(* CODESYS project Mahle_FilterLine_TempControl_17_01_20.project
   Title: Mahle_FilterLine_TempControl_03_01_20
   Version: 0.0.0.0

Project tree, tasks and I/O mapping:
  MyController : TM218LDAE24DRHN, Schneider Electric, order no. TM218LDAE24DRHN, version 4.0.1.26
      settings: Expansion Tasks.Expansion 1 Task Name = 'MAST'
    application Application
      libraries: Standard, * (System)
      task MAST (cyclic, interval 20 ms, priority 15, watchdog 100 ms x 1) calls POU
      function HiddenPOU [ST]
      global variables GVL
      program POU [FBD]
      function block tempAvergaging [ST]
      function block tempController [ST]
      function block calculateCycleTime [ST]
      function CheckBounds [ST]
      function block pressureAlarm [ST]
    Embedded Functions
      IO : IO, Schneider Electric, version 4.0.1.26
          input  iwIO_IW0 : WORD  // IW0
          input  iAuto : BOOL  // IW0.I0
          input  iPanelPB : BOOL  // IW0.I1
          input  iStartPB : BOOL  // IW0.I2
          input  iStopPB : BOOL  // IW0.I3
          input  iThyristorTrip : BOOL  // IW0.I6
          input  iFwdSensor : BOOL  // IW0.I8
          output qStartMC : BOOL  // QW0.Q0
          output qHeaterDown : BOOL  // QW0.Q1
          output qYellow : BOOL  // QW0.Q2
          output qGreen : BOOL  // QW0.Q3
          output qRed : BOOL  // QW0.Q4
          output qHooter : BOOL  // QW0.Q5
          unmapped channels: QW0
      HSC : HSC, Schneider Electric, version 4.0.1.26
    Serial Line 1
      SoMachine_Network_Manager : SoMachine-Network Manager, Schneider Electric, version 4.0.0.2
    Serial Line 2
      Modbus_Manager : Modbus Manager, Schneider Electric, version 4.0.0.2
    Ethernet
        settings: IPAddress = [192, 168, 1, 1]; SubnetMask = [255, 255, 255, 0]; WebServer = FALSE; FTP Server = FALSE; SoMachine Protocol = TRUE; Modbus Server = TRUE; NetManage Protocol = FALSE; SNMP protocol = FALSE; Enable Routing = FALSE
    Module_1 : TM2AMM3HT, Schneider Electric, order no. TM2AMM3HT, version 4.0.1.26
        settings: IW0.Maximum = 4000; IW1.Maximum = 1000; QW0.Maximum = 1000
        input  iwTempSensor : INT  // IW0
        input  iwPressureSensor : INT  // IW1
        output qwHeater : INT  // QW0
*)

// MyController/Application/GVL
VAR_GLOBAL
	thyristorTrip AT %MX600.0: BOOL;
	autoSel AT %MX600.1: BOOL;
	mcRunning AT %MX600.2: BOOL;
	heaterDown AT %MX600.3: BOOL;
	startSensing AT %MX600.4: BOOL;
	pressureLow AT %MX600.5: BOOL;
	resetPressMinMax AT %MX600.6: BOOL;
	cycleError AT %MX600.7: BOOL;
	startMCRun: BOOL;
	
	pressLowAlarm: BOOL;
	pressHighAlarm: BOOL;
END_VAR
VAR_GLOBAL RETAIN
	tempOffset AT %MD0: REAL :=0;
	puckTemp AT %MD1: REAL;
	finalCount AT %MD2: DINT;
	propGain AT %MD3: REAL;
	integGain AT %MD4: REAL;
	derivative AT %MD5: REAL;
	setTemp AT %MD6: REAL :=195;
	puckTempAvg AT %MD7: REAL;
	heaterManualSP AT %MD8: REAL :=50;
	heaterPIDOut AT %MD9: REAL;
	
	cycleTime AT %MD10: REAL;
	timeBWPucks AT %MD11: REAL;
	heaterLowRun AT %MD12: REAL :=48;
	heaterHighRun AT %MD13: REAL :=55;
	
	pressure AT %MD14: REAL;
	pressHighSet AT %MD15: REAL;
	pressLowSet AT %MD16: REAL;
	pressMin AT %MD17: REAL;
	pressMax AT %MD18: REAL;	
	pressureOffset AT %MD19: REAL;
	AvgPressure AT %MD21: REAL;
	
	startDelay AT %MW100: INT :=6;
	mcStopTime AT %MW101: INT :=30;
	pressAlarmDelay AT %MW102: INT;
	
	heaterManualOn AT %MX602.0: BOOL;
	heaterManualDown AT %MX602.1: BOOL;
	
END_VAR

// MyController/Application/POU
PROGRAM POU
VAR
	puckTemp1: REAL;
	tempAvergaging_0: tempAvergaging;
	PID_0: PID;
	RS_0: RS;
	runMC: BOOL;
	R_TRIG_0: R_TRIG;
	PID_1: PID_FIXCYCLE;
	TON_0: TON;
	tempController_0: tempController;
	TP_0: TP;
	mcStartDelayTime: TIME;
	TON_1: TON;
	calculateCycleTime_0: calculateCycleTime;
	sensorTrig: BOOL;
	TP_1: TP;
	stopTime: TIME;
	TON_2: TON;
	stopTimeET: TIME;
	stopHeater: BOOL;
	pressureAlarm_0: pressureAlarm;
	pressAlarm: BOOL;
	startProduction: BOOL;
	greenCont: BOOL;
	BLINK_0: BLINK;
	BLINK_1: BLINK;
	stopHeater1: BOOL;
	RS_1: RS;
END_VAR

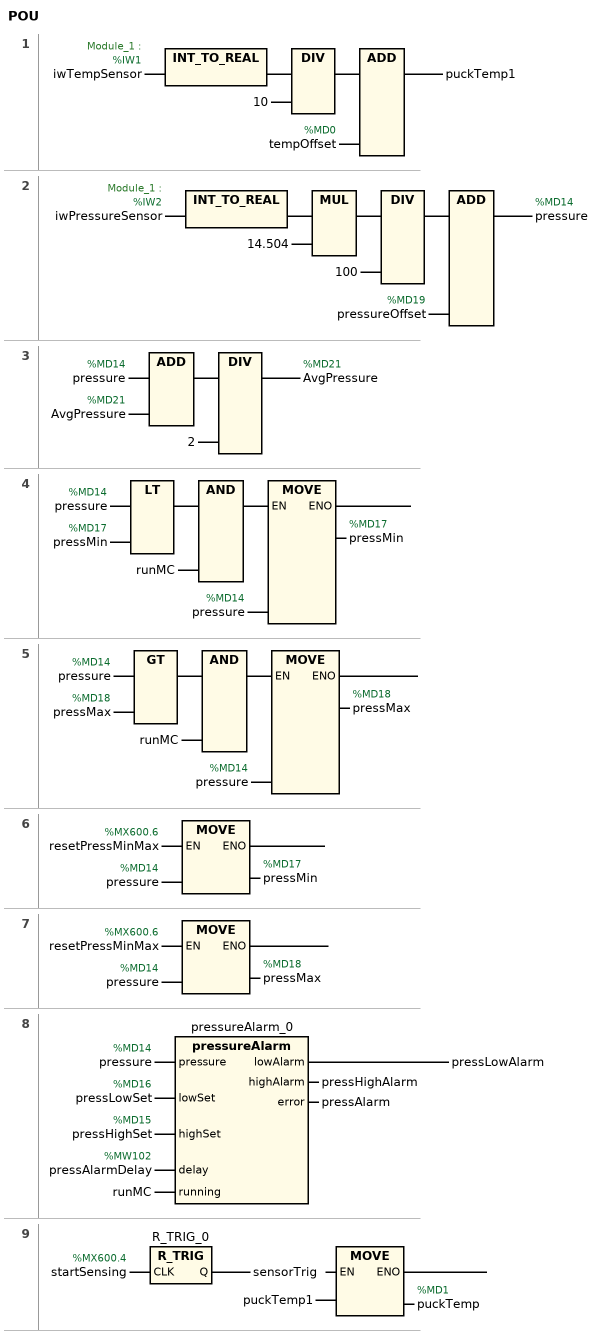
// NETWORK 1
//   iwTempSensor: Module_1 : | AT %IW1
//   tempOffset: AT %MD0
puckTemp1 := INT_TO_REAL(iwTempSensor) / 10 + tempOffset;

// NETWORK 2
//   iwPressureSensor: Module_1 : | AT %IW2
//   pressureOffset: AT %MD19
//   pressure: AT %MD14
pressure := (INT_TO_REAL(iwPressureSensor) * 14.504) / 100 + pressureOffset;

// NETWORK 3
//   pressure: AT %MD14
//   AvgPressure: AT %MD21
AvgPressure := (pressure + AvgPressure) / 2;

// NETWORK 4
//   pressure: AT %MD14
//   pressMin: AT %MD17
IF pressure < pressMin AND runMC THEN pressMin := pressure; END_IF

// NETWORK 5
//   pressure: AT %MD14
//   pressMax: AT %MD18
IF pressure > pressMax AND runMC THEN pressMax := pressure; END_IF

// NETWORK 6
//   resetPressMinMax: AT %MX600.6
//   pressure: AT %MD14
//   pressMin: AT %MD17
IF resetPressMinMax THEN pressMin := pressure; END_IF

// NETWORK 7
//   resetPressMinMax: AT %MX600.6
//   pressure: AT %MD14
//   pressMax: AT %MD18
IF resetPressMinMax THEN pressMax := pressure; END_IF

// NETWORK 8
//   pressure: AT %MD14
//   pressLowSet: AT %MD16
//   pressHighSet: AT %MD15
//   pressAlarmDelay: AT %MW102
pressureAlarm_0(
    pressure := pressure,
    lowSet := pressLowSet,
    highSet := pressHighSet,
    delay := pressAlarmDelay,
    running := runMC,
    highAlarm => pressHighAlarm,
    error => pressAlarm); // pressureAlarm
pressLowAlarm := pressureAlarm_0.lowAlarm;

// NETWORK 9
//   startSensing: AT %MX600.4
//   puckTemp: AT %MD1
R_TRIG_0(CLK := startSensing); // R_TRIG
sensorTrig := R_TRIG_0.Q;
IF R_TRIG_0.Q THEN puckTemp := puckTemp1; END_IF

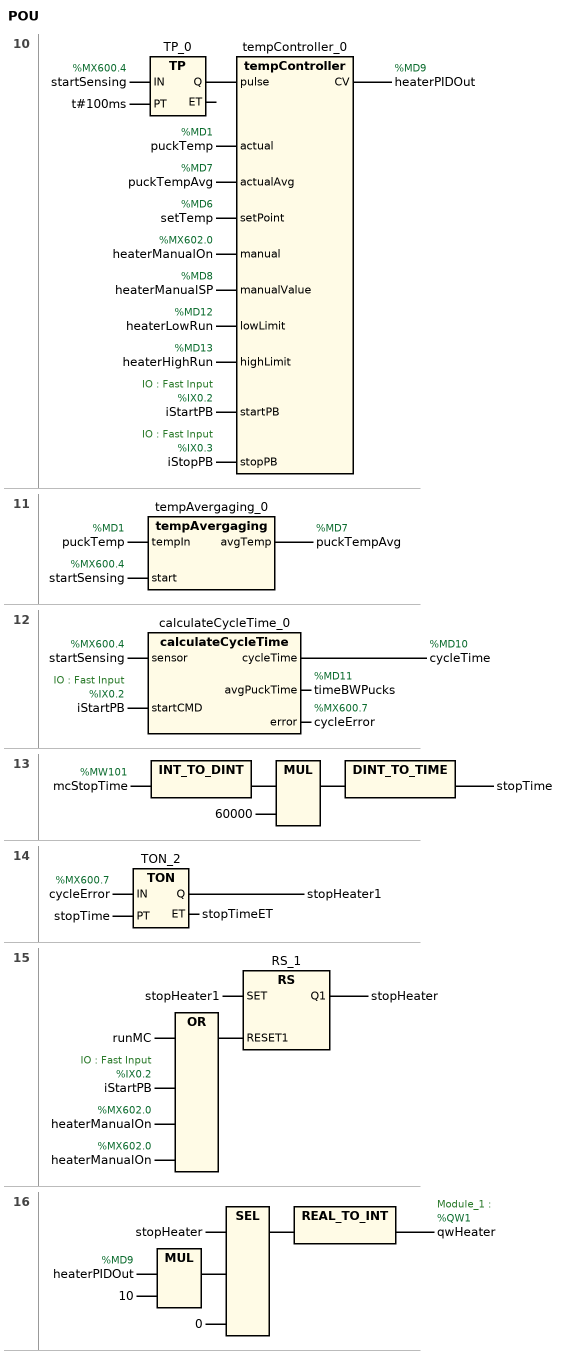
// NETWORK 10
//   startSensing: AT %MX600.4
//   puckTemp: AT %MD1
//   puckTempAvg: AT %MD7
//   setTemp: AT %MD6
//   heaterManualOn: AT %MX602.0
//   heaterManualSP: AT %MD8
//   heaterLowRun: AT %MD12
//   heaterHighRun: AT %MD13
//   iStartPB: IO : Fast Input | AT %IX0.2
//   iStopPB: IO : Fast Input | AT %IX0.3
//   heaterPIDOut: AT %MD9
TP_0(IN := startSensing, PT := t#100ms); // TP
tempController_0(
    pulse := TP_0.Q,
    actual := puckTemp,
    actualAvg := puckTempAvg,
    setPoint := setTemp,
    manual := heaterManualOn,
    manualValue := heaterManualSP,
    lowLimit := heaterLowRun,
    highLimit := heaterHighRun,
    startPB := iStartPB,
    stopPB := iStopPB); // tempController
heaterPIDOut := tempController_0.CV;

// NETWORK 11
//   puckTemp: AT %MD1
//   startSensing: AT %MX600.4
//   puckTempAvg: AT %MD7
tempAvergaging_0(tempIn := puckTemp, start := startSensing); // tempAvergaging
puckTempAvg := tempAvergaging_0.avgTemp;

// NETWORK 12
//   startSensing: AT %MX600.4
//   iStartPB: IO : Fast Input | AT %IX0.2
//   timeBWPucks: AT %MD11
//   cycleError: AT %MX600.7
//   cycleTime: AT %MD10
calculateCycleTime_0(
    sensor := startSensing,
    startCMD := iStartPB,
    avgPuckTime => timeBWPucks,
    error => cycleError); // calculateCycleTime
cycleTime := calculateCycleTime_0.cycleTime;

// NETWORK 13
//   mcStopTime: AT %MW101
stopTime := DINT_TO_TIME(INT_TO_DINT(mcStopTime) * 60000);

// NETWORK 14
//   cycleError: AT %MX600.7
TON_2(IN := cycleError, PT := stopTime, ET => stopTimeET); // TON
stopHeater1 := TON_2.Q;

// NETWORK 15
//   iStartPB: IO : Fast Input | AT %IX0.2
//   heaterManualOn: AT %MX602.0
RS_1(SET := stopHeater1, RESET1 := runMC OR iStartPB OR heaterManualOn OR heaterManualOn); // RS
stopHeater := RS_1.Q1;

// NETWORK 16
//   heaterPIDOut: AT %MD9
//   qwHeater: Module_1 : | AT %QW1
qwHeater := REAL_TO_INT(SEL(stopHeater, heaterPIDOut * 10, 0));

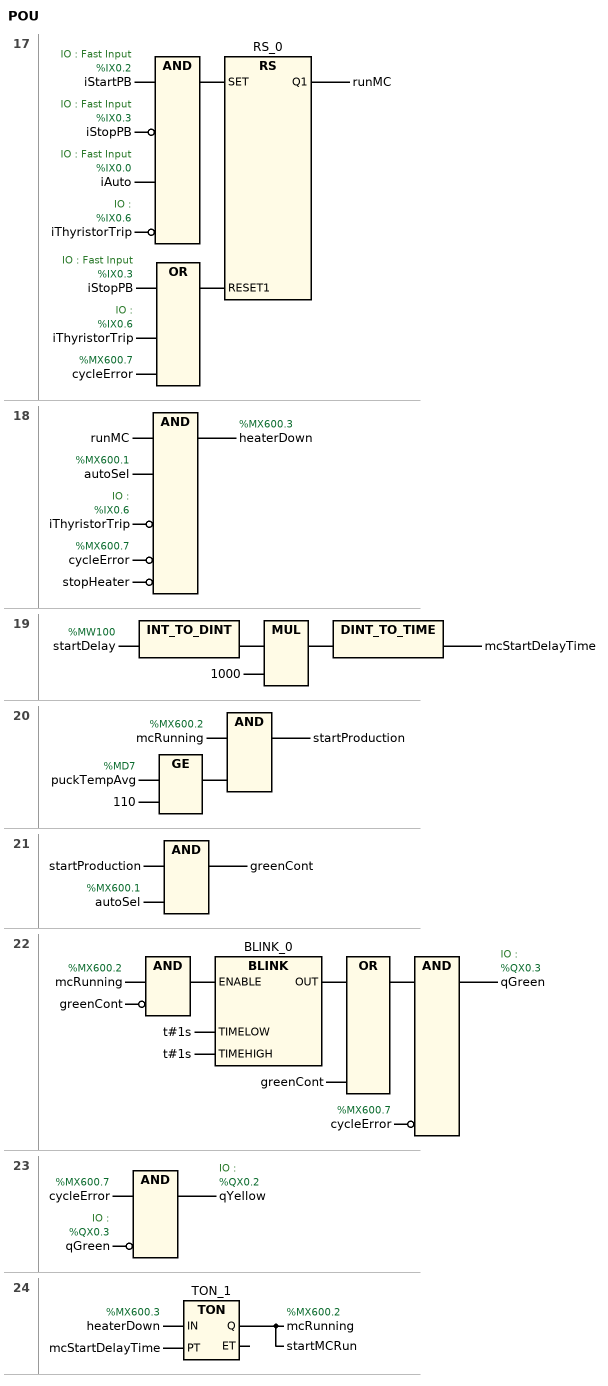
// NETWORK 17
//   iStartPB: IO : Fast Input | AT %IX0.2
//   iStopPB: IO : Fast Input | AT %IX0.3
//   iAuto: IO : Fast Input | AT %IX0.0
//   iThyristorTrip: IO : | AT %IX0.6
//   cycleError: AT %MX600.7
RS_0(SET := iStartPB AND NOT iStopPB AND iAuto AND NOT iThyristorTrip, RESET1 := iStopPB OR iThyristorTrip OR cycleError); // RS
runMC := RS_0.Q1;

// NETWORK 18
//   autoSel: AT %MX600.1
//   iThyristorTrip: IO : | AT %IX0.6
//   cycleError: AT %MX600.7
//   heaterDown: AT %MX600.3
heaterDown := runMC AND autoSel AND NOT iThyristorTrip AND NOT cycleError AND NOT stopHeater;

// NETWORK 19
//   startDelay: AT %MW100
mcStartDelayTime := DINT_TO_TIME(INT_TO_DINT(startDelay) * 1000);

// NETWORK 20
//   mcRunning: AT %MX600.2
//   puckTempAvg: AT %MD7
startProduction := mcRunning AND puckTempAvg >= 110;

// NETWORK 21
//   autoSel: AT %MX600.1
greenCont := startProduction AND autoSel;

// NETWORK 22
//   mcRunning: AT %MX600.2
//   cycleError: AT %MX600.7
//   qGreen: IO : | AT %QX0.3
BLINK_0(ENABLE := mcRunning AND NOT greenCont, TIMELOW := t#1s, TIMEHIGH := t#1s); // BLINK
qGreen := (BLINK_0.OUT OR greenCont) AND NOT cycleError;

// NETWORK 23
//   cycleError: AT %MX600.7
//   qGreen: IO : | AT %QX0.3
//   qYellow: IO : | AT %QX0.2
qYellow := cycleError AND NOT qGreen;

// NETWORK 24
//   heaterDown: AT %MX600.3
//   mcRunning: AT %MX600.2
TON_1(IN := heaterDown, PT := mcStartDelayTime); // TON
mcRunning := TON_1.Q;
startMCRun := TON_1.Q;

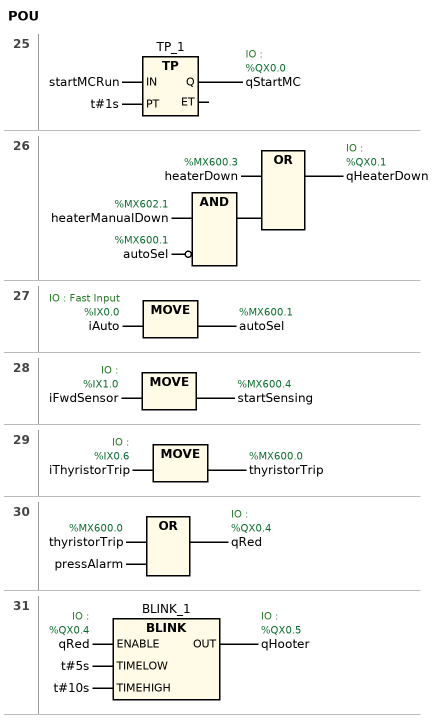
// NETWORK 25
//   qStartMC: IO : | AT %QX0.0
TP_1(IN := startMCRun, PT := t#1s); // TP
qStartMC := TP_1.Q;

// NETWORK 26
//   heaterDown: AT %MX600.3
//   heaterManualDown: AT %MX602.1
//   autoSel: AT %MX600.1
//   qHeaterDown: IO : | AT %QX0.1
qHeaterDown := heaterDown OR heaterManualDown AND NOT autoSel;

// NETWORK 27
//   iAuto: IO : Fast Input | AT %IX0.0
//   autoSel: AT %MX600.1
autoSel := iAuto;

// NETWORK 28
//   iFwdSensor: IO : | AT %IX1.0
//   startSensing: AT %MX600.4
startSensing := iFwdSensor;

// NETWORK 29
//   iThyristorTrip: IO : | AT %IX0.6
//   thyristorTrip: AT %MX600.0
thyristorTrip := iThyristorTrip;

// NETWORK 30
//   thyristorTrip: AT %MX600.0
//   qRed: IO : | AT %QX0.4
qRed := thyristorTrip OR pressAlarm;

// NETWORK 31
//   qRed: IO : | AT %QX0.4
//   qHooter: IO : | AT %QX0.5
BLINK_1(ENABLE := qRed, TIMELOW := t#5s, TIMEHIGH := t#10s); // BLINK
qHooter := BLINK_1.OUT;

END_PROGRAM

// MyController/Application/pressureAlarm
FUNCTION_BLOCK pressureAlarm
VAR_INPUT
	pressure: REAL;
	lowSet: REAL;
	highSet: REAL;
	delay: INT;
	running: BOOL;
END_VAR
VAR_OUTPUT
	lowAlarm: BOOL;
	highAlarm: BOOL;
	error: BOOL;
END_VAR
VAR
	timeDelay: TIME;
	startTON1: BOOL;
	startTON2: BOOL;
	TON1: TON;
	TON2: TON;
END_VAR

timeDelay := DINT_TO_TIME(INT_TO_DINT(delay)*1000);

TON1(IN:=startTON1, PT:=timeDelay);
TON2(IN:=startTON2, PT:=timeDelay);

IF running THEN
	IF pressure < lowSet THEN
		startTON1 := TRUE;
	ELSE
		startTON1 := FALSE;
	END_IF

	IF pressure > highSet THEN
		startTON2 := TRUE;
	ELSE
		startTON2 := FALSE;
	END_IF			
	
	IF ton1.Q THEN
		lowAlarm := TRUE;
	ELSE
		lowAlarm := FALSE;
	END_IF
	
	IF ton2.Q THEN
		highAlarm := TRUE;
	ELSE
		highAlarm := FALSE;
	END_IF
	
	IF lowAlarm OR highAlarm THEN
		error := TRUE;
	ELSE
		error := FALSE;
	END_IF
END_IF

END_FUNCTION_BLOCK

// MyController/Application/tempController
FUNCTION_BLOCK tempController
VAR_INPUT
	pulse: BOOL;
	actual: REAL;
	actualAvg: REAL;
	setPoint: REAL;
	manual: BOOL;
	manualValue: REAL;
	lowLimit: REAL;
	highLimit: REAL;
	startPB: BOOL;
	stopPB: BOOL;
END_VAR
VAR_OUTPUT
	CV: REAL;
END_VAR
VAR
	error: REAL;
	errorPC: REAL;
	CV1: REAL;
	errorPCAbs: REAL;
	errorFromAvg: REAL;
	startHeater: BOOL;
	CV2: REAL;
END_VAR

IF startPB AND NOT manual THEN
	startHeater := TRUE;
	CV1 := highLimit;
END_IF
IF pulse AND NOT manual THEN
	error := setPoint - actual;
	errorPC := (error*100)/setPoint;
	errorFromAvg := actualAvg - actual;
	IF errorFromAvg < 20 AND errorFromAvg > -20 THEN
	
		IF errorPC >=0 THEN
			errorPCAbs := errorPC;
		ELSE
			errorPCAbs := -1*errorPC;
		END_IF
	
		IF errorPCAbs < 2 THEN
			CV1 := CV+(errorPC/90);
		ELSIF errorPCAbs < 5 THEN
			CV1 := CV + (errorPC/50);
		ELSIF errorPCAbs < 15 THEN
			CV1 := CV + (errorPC/75);
		ELSE
			CV1 := CV + (errorPC/100);				
		END_IF
	END_IF
END_IF

IF manual THEN
	CV := manualValue;
ELSE
	CV := CV2;
END_IF

IF CV1 < lowLimit THEN
	CV2 := lowLimit;
ELSIF CV1 > highLimit THEN
	CV2 := highLimit;
ELSE
	CV2 := CV1;
END_IF

END_FUNCTION_BLOCK

// MyController/Application/tempAvergaging
FUNCTION_BLOCK tempAvergaging
VAR_INPUT
	tempIn: REAL;
	start: BOOL;
END_VAR
VAR_OUTPUT
	avgTemp: REAL;
END_VAR
VAR
	counter1: CTU;
	x1: REAL :=0;
	x2: REAL :=0;
	x3: REAL :=0;
	x4: REAL :=0;
	x5: REAL :=0;
	x6: REAL :=0;
	x7: REAL :=0;
	x8: REAL :=0;
	x9: REAL :=0;
	x10: REAL :=0;
	x11: REAL :=0;
	x12: REAL :=0;
	countReset: BOOL;
END_VAR

counter1(CU:=start, RESET:=countReset, PV:=5);
CASE counter1.CV OF
	1:	x1:=tempIn;
	2:	x2:=tempIn;
	3:	x3:=tempIn;
	4:	x4:=tempIn;
	5:	x5:=tempIn;
//	6:	x6:=tempIn;
//	7:	x7:=tempIn;
//	8:	x8:=tempIn;
//	9:	x9:=tempIn;
//	10:	x10:=tempIn;
//	11:	x11:=tempIn;
//	12:	x12:=tempIn;
END_CASE

IF counter1.Q THEN
	countReset := TRUE;
ELSE
	countReset := FALSE;
END_IF

//avgTemp := (x1+x2+x3+x4+x5+x6+x7+x8+x9+x10+x11+x12)/12;

avgTemp := (x1+x2+x3+x4+x5)/5;

END_FUNCTION_BLOCK

// MyController/Application/calculateCycleTime
FUNCTION_BLOCK calculateCycleTime
VAR_INPUT
	sensor: BOOL;
	startCMD: BOOL;
END_VAR
VAR_OUTPUT
	cycleTime: REAL;
	avgPuckTime: REAL;
	error: BOOL;
END_VAR
VAR
	ton1: TON;
	ton2: TON;
	ton3: TON;
	ctu1: CTU;
	ctu2: CTU;
	ctuReset: BOOL;
	startTON1: BOOL;
	startTON2: BOOL;
	startTON3: BOOL;
	startTON4: BOOL;
	t1Time: REAL;
	t2Time: REAL;
	t3Time: REAL;
	t4Time: REAL;
	ctuReset2: BOOL;
	t1: REAL;
	t2: REAL;
	t3: REAL;
	t4: REAL;
	t5: REAL;
	t6: REAL;
	t7: REAL;
	t8: REAL;
	t9: REAL;
	t10: REAL;
	t11: REAL;
	t12: REAL;
	t13: REAL;
	t14: REAL;
	t15: REAL;
	t16: REAL;
	t17: REAL;
	t18: REAL;
	t19: REAL;
	t20: REAL;
	t21: REAL;
	t22: REAL;
	t23: REAL;
	t24: REAL;
	firstRun: BOOL;
	ton4: TON;
	ton5: TON;
	newCycleStart: BOOL;
	rtrig1: R_TRIG;
	rtrig2: R_TRIG;
	trig2: BOOL;
	t1TimeInit: REAL;
	t2TimeInit: REAL;
	ctu3: CTU;
	cycleDone: BOOL;
	ctu3Reset: BOOL;
	t4TimeInit: REAL;
	t3TimeInit: REAL;
	tof1: TOF;
END_VAR


	
ctu1(CU:=sensor, RESET:=ctuReset, PV:=2);
ton1(IN:=startTON1, PT:=T#30M);
ton2(IN:=startTON2, PT:=T#30M);
ton3(IN:=startTON3, PT:=T#60M);
ton4(IN:=startTON4, PT:=T#60M);
ton5(IN:=newCycleStart, PT:=T#100MS);
ctu2(CU:=sensor, RESET:=ctu2.Q, PV:=24);
ctu3(CU:=cycleDone, RESET:=ctu3Reset, PV:=2);
tof1(IN:=startCMD, PT:=T#30S);

	IF ctu1.CV = 1 THEN
		startTON1 := TRUE;
		startTON2:= FALSE;	
		t2Time := t2TimeInit;
	END_IF

	IF ctu1.CV = 2 THEN
		startTON1:=FALSE;
		startTON2:= TRUE;
		t1Time := t1TimeInit;
	END_IF
	
	IF ctu1.CV >= 2 THEN
		ctuReset := TRUE;
	ELSE	
		ctuReset := FALSE;
	END_IF

	IF startTON1 THEN
		t1TimeInit := TIME_TO_REAL(ton1.ET);
	END_IF

	IF startTON2 THEN
		t2TimeInit := TIME_TO_REAL(ton2.ET);
	END_IF

	CASE ctu2.CV OF
		2:	t1:=t1Time;
		3:	t2:=t2Time;
		4:	t3:=t1Time;
		5:	t4:=t2Time;
		6:	t5:=t1Time;
		7:	t6:=t2Time;
		8:	t7:=t1Time;
		9:	t8:=t2Time;
		10:	t9:=t1Time;
		11:	t10:=t2Time;
		12:	t11:=t1Time;
		13:	t12:=t2Time;
		14:	t13:=t1Time;
		15:	t14:=t2Time;
		16:	t15:=t1Time;
		17:	t16:=t2Time;
		18:	t17:=t1Time;
		19:	t18:=t2Time;
		20:	t19:=t1Time;
		21:	t20:=t2Time;
		22:	t21:=t1Time;
		23:	t22:=t2Time;
		0:	t23:=t1Time;
		1:	t24:=t2Time;
	END_CASE
		
	IF TIME_TO_REAL(ton1.ET) > (avgPuckTime*1000+4000) AND NOT tof1.Q THEN
		error := TRUE;
	ELSIF TIME_TO_REAL(ton2.ET) > (avgPuckTime*1000+4000)  AND NOT tof1.Q THEN
		error := TRUE;
	ELSE
		error := FALSE;
	END_IF
	
	IF startTON3 THEN
		t3TimeInit := TIME_TO_REAL(ton3.ET);
	END_IF
	IF startTON4 THEN
		t4TimeInit := TIME_TO_REAL(ton4.ET);
	END_IF

	IF ctu2.CV = 1 THEN
		cycleDone := TRUE;
	ELSE
		cycleDone := FALSE;
	END_IF
	
	IF ctu3.CV = 1 THEN
		startTON3 := TRUE;
		startTON4:= FALSE;	
		t4Time := t4TimeInit;
	END_IF

	IF ctu3.CV = 2 THEN
		startTON3:=FALSE;
		startTON4:= TRUE;
		t3Time := t3TimeInit;
	END_IF
	
	IF ctu3.CV >= 2 THEN
		ctu3Reset := TRUE;
	ELSE	
		ctu3Reset := FALSE;
	END_IF
	
	IF NOT error THEN
		avgPuckTime := (t1+t2+t3+t4+t5+t6+t7+t8+t9+t10+t11+t12+t13+t14+t15+t16+t17+t18+t19+t20+t21+t22+t23+t24)/24000;
		cycleTime := (t3Time+t4Time)/2000;
	END_IF

END_FUNCTION_BLOCK

// MyController/Application/HiddenPOU
FUNCTION HiddenPOU : BOOL

VAR_INPUT
	pHiddenFunc: POINTER TO WORD;
END_VAR
VAR
	pRead: POINTER TO BYTE;
	pWrite: POINTER TO BYTE;
END_VAR

pRead := pHiddenFunc + 400;
pWrite := pHiddenFunc + 4400;
HiddenPOU := TRUE;

END_FUNCTION

// MyController/Application/CheckBounds
// Implicitly generated code : DO NOT EDIT
FUNCTION CheckBounds : DINT
VAR_INPUT
	index, lower, upper: DINT;
END_VAR

// Implicitly generated code : Only an Implementation suggestion
IF  index < lower THEN
	CheckBounds := lower;
ELSIF  index > upper THEN
	CheckBounds := upper;
ELSE  
	CheckBounds := index;
END_IF

END_FUNCTION
